FUNCTION_BLOCK INTERNAL FB_DischargeState IMPLEMENTS I_State
VAR
	pMachine		: POINTER TO FB_Machine; // Points to the state machine (THIS)
	fVSensors		: ARRAY [0..1] OF REAL; 
END_VAR

METHOD PUBLIC Check
VAR
	fLoadVoltage			: REAL; 
	fInputVoltage			: REAL; 
END_VAR
THIS^.ResetContactors(); // THE CONTACTORS NEED TO ALAWAYS BE OPEN IN THIS STATE NO MATTER WHAT WAS THE PREVIOUS STATE
THIS^.ResetTimer(); // in case the emergency stop is pressed while the circuit is in precharge state
fVSensors := THIS^.pMachine^.VSensors;

fInputVoltage := fVSensors[0];
fLoadVoltage := fVSensors[1];

IF (fLoadVoltage < 0.1 * fInputVoltage) THEN
	THIS^.pMachine^.Message := '[DISCHARGE] The load voltage is now less than 1 percent of the input voltage.$0A WAITING FOR ACKNOWLEDGEMENT TO DISCONNECT SYSTEM.';
ELSE 
	THIS^.pMachine^.Message := '[DISCHARGE] Waiting for load voltage to be lower than 10 percent of the input voltage.';
END_IF
END_METHOD

PROPERTY PUBLIC Description : STRING
GET
Description := 'DISCHARGE';
END_GET
END_PROPERTY

METHOD PUBLIC FB_init
VAR_INPUT
	bInitRetains : BOOL; // if TRUE, the retain variables are initialized (warm start / cold start)
	bInCopyCode : BOOL;  // if TRUE, the instance afterwards gets moved into the copy code (online change)
	pMachine		: POINTER TO FB_Machine; // Points to the state machine (THIS)
END_VAR
THIS^.pMachine := pMachine;
END_METHOD

METHOD PUBLIC PressButton 
VAR
	fLoadVoltage		: REAL; 
	fInputVoltage		: REAL; 
END_VAR
fVSensors := THIS^.pMachine^.VSensors;
fInputVoltage := fVSensors[0];
fLoadVoltage := fVSensors[1];

IF (fLoadVoltage < 0.1 * fInputVoltage) THEN
	THIS^.pMachine^.Message := '[DISCHARGE] Acknowledge button has been pressed. $0A SYSTEM ENTERS DISCONNECTED STATE.';
	THIS^.pMachine^.SetState(THIS^.pMachine^.DisconnectedState);
END_IF
END_METHOD

METHOD PUBLIC PressDischarge
END_METHOD

METHOD PUBLIC Reset
END_METHOD

METHOD PUBLIC ResetContactors
VAR
	nIdx					: INT := 0; 
	bBypassContactors		: ARRAY[0..1] OF BOOL; 
	bMainContactors			: ARRAY[0..1] OF BOOL; 
END_VAR
FOR nIdx := 0 TO 1 BY 1 DO 
	bBypassContactors[nIdx] := FALSE;
	bMainContactors[nIdx] := FALSE; 
END_FOR

THIS^.pMachine^.BypassContactors := bBypassContactors; // Reset every contactor 
THIS^.pMachine^.MainContactors := bMainContactors;
END_METHOD

METHOD PUBLIC ResetTimer
THIS^.pMachine^.charge_TON.IN := FALSE;
END_METHOD

METHOD PUBLIC Stop
THIS^.pMachine^.SetState(THIS^.pMachine^.ErrorState);
END_METHOD

METHOD PUBLIC TimerDone
END_METHOD

END_FUNCTION_BLOCK

(* stored: Version 1.1.0.1, ProductVersion 3.1.4024.12
   POU FB_DischargeState: Id {d936db11-0e95-46d7-81bd-179f7d572f5f}, SpecialFunc None
   Method Check: Id {e77e82bd-9732-4d14-97e6-f45fe3cbee73}
   Property Description: Id {10b747bc-a5f5-42e4-9e65-f99c74376d25}
   Get Get: Id {ea3a037d-09e6-4763-a38c-ac1899021b9a}
   Method FB_init: Id {ee9d4094-8995-41ea-a6eb-751972b2dceb}
   Method PressButton: Id {4b95c776-2eae-4fd5-a550-441e9aa9038d}
   Method PressDischarge: Id {48a24bc7-2eef-49e1-ad6f-c16283f46719}
   Method Reset: Id {1c6d2c1d-ccf5-42f4-9d9e-e8be902f80bc}
   Method ResetContactors: Id {9e9d5034-c6a6-4e71-9ab9-f9a397f67841}
   Method ResetTimer: Id {76b95b83-b0d7-40ca-af06-4cb9bb2aac1d}
   Method Stop: Id {ae487eac-c183-44d2-9ed6-5dcf1898df87}
   Method TimerDone: Id {9b1c3bd0-4a2f-4498-8236-60f3b0455476} *)
